DATA_BLOCK "ST10_Flow3_A1RotaryScan_iDB"
{ S7_Optimized_Access := 'TRUE' }
VERSION : 0.1
NON_RETAIN
// ATTRIBUTES
// AUTO_NUMBER = False
// BLOCK_NUMBER = 1073
// END_ATTRIBUTES
"ST10_Flow3_A1RotaryShaftScan"

BEGIN

END_DATA_BLOCK

